INTERFACE I_MotionAxis EXTENDS __SYSTEM.IQueryInterface, 
// 						I_AxisParameters, 
// 						I_AxisStatus, 
// 						I_Home,
// 						I_Halt, 
// 						I_Power, 
// 						I_Reset,
 						I_Output
// 						I_MoveAbsolute,
// 						I_BacklashCompensation

PROPERTY AbortDone : BOOL
GET
END_GET
END_PROPERTY

METHOD AxisEnabled : BOOL
VAR_INPUT
END_VAR
END_METHOD

PROPERTY AxisParamsInit : BOOL
GET
END_GET
END_PROPERTY

PROPERTY AxisState : MC_AxisStates
GET
END_GET
END_PROPERTY

(*
    Handle positive/negative backlash compensation
    User needs to set the direction of backlash from the sign of the compensation value
    Backlash compensation is disabled during referencing (homing).
    When direction is positive/negative, further movement in the negative/positive direction not compensated
    further movement in the negative/positive direction will be compensated
*)
METHOD BacklashCompensation
VAR_INPUT
    Active     : BOOL;
    Compensation	: LREAL;
    RampVelocity	: LREAL;
    DisableMode	: E_DISABLEMODE := E_DISABLEMODE.DisableModeHold;
END_VAR
END_METHOD

(*synced Fbs need just to activate the compensation with a given ramp speed
  other parameters are provided via EPICS (declared in this FB) or via the more extended BackalshCompensation method (simulation) *)
METHOD BacklashCompensationActive
VAR_INPUT
    Active     : BOOL;
    RampVelocity : LREAL;
END_VAR
END_METHOD

{warning 'Add property implementation'}
PROPERTY BacklashCompStatus : BOOL
GET
END_GET
END_PROPERTY

PROPERTY BacklashCompUserEn : BOOL
SET
END_SET
END_PROPERTY

METHOD Halt
VAR_INPUT
	Execute : BOOL;
    Deceleration : LREAL := 0.0;
    Jerk : LREAL := 0.0;
    BufferMode	: MC_BufferMode := MC_BufferMode.MC_Aborting;
END_VAR
END_METHOD

{warning 'Add property implementation'}
PROPERTY HaltActive : BOOL
GET
END_GET
END_PROPERTY

PROPERTY HaltBusy : BOOL
GET
END_GET
END_PROPERTY

PROPERTY HaltDone : BOOL
GET
END_GET
END_PROPERTY

METHOD  Home
VAR_INPUT
	Execute	: BOOL;
	HomeSpeedFast	: LREAL;
	HomeSpeedSlow	: LREAL;
END_VAR
END_METHOD

PROPERTY HomeBusy : BOOL
GET
END_GET
END_PROPERTY

PROPERTY HomeDone : BOOL
GET
END_GET
END_PROPERTY

PROPERTY HomeMode : E_EpicsHomeCmd
GET
END_GET
SET
END_SET
END_PROPERTY

PROPERTY InTargetPosition : BOOL
GET
END_GET
END_PROPERTY

{warning 'Add property implementation'}
PROPERTY MeasureBacklash : LREAL
GET
END_GET
END_PROPERTY

PROPERTY MeasuredAcceleration : LREAL
GET
END_GET
END_PROPERTY

{warning 'Add property implementation'}
PROPERTY MeasuredBacklashComp : LREAL
GET
END_GET
END_PROPERTY

PROPERTY MeasuredPosition : LREAL
GET
END_GET
END_PROPERTY

PROPERTY MeasuredPositionDiff : LREAL
GET
END_GET
END_PROPERTY

PROPERTY MeasuredVelocity : LREAL
GET
END_GET
END_PROPERTY

METHOD MoveAbsolute
VAR_INPUT
    Execute     : BOOL;
    Position	: LREAL;
    Velocity	: LREAL;
    Acceleration	: LREAL := 0.0;
    Deceleration	: LREAL := 0.0;
    Jerk	: LREAL := 0.0;
    BufferMode	: MC_BufferMode := MC_BufferMode.MC_Aborting;
END_VAR
END_METHOD

PROPERTY MoveAbsoluteAborted : BOOL
GET
END_GET
END_PROPERTY

PROPERTY MoveAbsoluteActive : BOOL
GET
END_GET
END_PROPERTY

PROPERTY MoveAbsoluteBusy : BOOL
GET
END_GET
END_PROPERTY

PROPERTY MoveAbsoluteDone : BOOL
GET
END_GET
END_PROPERTY

PROPERTY NegativeMotionIsEnabled : BOOL
GET
END_GET
END_PROPERTY

PROPERTY PositiveMotionIsEnabled : BOOL
GET
END_GET
END_PROPERTY

METHOD Power
VAR_INPUT
    Enable	: BOOL;
    Enable_Positive	: BOOL;
    Enable_Negative	: BOOL;
    Override	: LREAL ;
    BufferMode	: MC_BufferMode;
END_VAR
END_METHOD

PROPERTY PowerActive : BOOL
GET
END_GET
END_PROPERTY

METHOD PowerEnables
VAR_INPUT
    Enable	: BOOL;
    Enable_Positive	: BOOL;
    Enable_Negative	: BOOL;
END_VAR
END_METHOD

PROPERTY PowerIsEnabled : BOOL
GET
END_GET
END_PROPERTY

METHOD Reset
VAR_INPUT
	Execute : BOOL;
END_VAR
END_METHOD

PROPERTY ResetBusy : BOOL
GET
END_GET
END_PROPERTY

PROPERTY ResetDone : BOOL
GET
END_GET
END_PROPERTY

PROPERTY RestoreDone : BOOL
GET
END_GET
END_PROPERTY

PROPERTY SavedPosition : LREAL
GET
END_GET
END_PROPERTY

PROPERTY ScaledEncoderCount : UDINT
GET
END_GET
END_PROPERTY

{warning 'Add property implementation'}
PROPERTY StandStill : BOOL
GET
END_GET
END_PROPERTY

(*
    Check all post condition before updating bCommandedMoveAbsolute
    The implmentatation will depend on the axis type
    DS402 NC/Direct axis : Implementation need to check that the drive is in the correct mode before initaiting the move then set bCommandedMoveAbsolute
    MP NC axis : will immediately write to bCommandedMoveAbsolute
*)
METHOD StartMove : BOOL
VAR_INPUT
    MoveMode	: E_EpicsMotorCmd;
    CmdExecute	: BOOL;
END_VAR
END_METHOD

PROPERTY Stopped : BOOL
GET
END_GET
END_PROPERTY

END_INTERFACE

(* stored: Version 1.1.0.1
   Itf I_MotionAxis: Id {31a902d0-0933-4477-af85-d5a81bbd2467}
   Property AbortDone: Id {5c7662f1-9d2d-42f7-8e24-51d5866c86b3}
   Get Get: Id {93658730-1b85-4a95-9fa2-c21fbe9d7f48}
   Method AxisEnabled: Id {65dbd00d-2aae-4126-bb1b-b72ba759e223}
   Property AxisParamsInit: Id {0ac6452c-b5e1-4e22-865e-3cb2fa5bdfa5}
   Get Get: Id {cf5c8d62-269a-4b22-88e4-cc443108703c}
   Property AxisState: Id {bff14cf8-c54e-4f81-89d2-2b0a7f44eac4}
   Get Get: Id {449be078-56bc-4849-bd3a-e15c9cea95eb}
   Method BacklashCompensation: Id {7436498c-944b-4e18-b9ff-6d68481a3f19}
   Method BacklashCompensationActive: Id {3e7bc661-61f7-4e53-a6c1-341c4d84a32c}
   Property BacklashCompStatus: Id {caf46bd6-b35f-44e4-8914-e70bbd07956d}
   Get Get: Id {f6a45633-a1fa-4659-887f-31976f0aa6aa}
   Property BacklashCompUserEn: Id {94812ccc-d5c4-49f8-aaf1-b91b9d04b484}
   Set Set: Id {84ab6711-b0cf-4074-b1dd-0d70c79947a1}
   Method Halt: Id {c05fa9c9-1bb9-49f8-8b3e-d44f26433d64}
   Property HaltActive: Id {5d6d5bda-e0de-4a28-8aa0-b85c507cdad0}
   Get Get: Id {4f5edcd4-20fe-43f9-8973-d65798036d1c}
   Property HaltBusy: Id {9541a085-e1d1-4a88-8402-724cd91f040a}
   Get Get: Id {8eb7f1c7-9461-46de-8fdb-d396cbb4626b}
   Property HaltDone: Id {a96c6505-72d4-48f7-834a-1162be0cc363}
   Get Get: Id {0d04f02a-d165-4498-8810-653cd0ad98be}
   Method Home: Id {389ec9c0-6958-4b75-bc75-cf73e213180f}
   Property HomeBusy: Id {085e184a-60b7-4e61-b9df-1cb084216a57}
   Get Get: Id {3e4fb446-eba9-4f63-a7ca-7692470d57ec}
   Property HomeDone: Id {180db6b4-ec37-4d47-b243-fc069ef95f8e}
   Get Get: Id {5abbdf75-4945-4b01-8731-586a4b17c65d}
   Property HomeMode: Id {82377409-78bc-42db-8154-8d4d5bb308ee}
   Get Get: Id {1a9eb16b-9f78-44c6-87e2-3304e572b793}
   Set Set: Id {6b7a652e-625f-499d-a110-8ca538ff003d}
   Property InTargetPosition: Id {01bb2d1f-6955-454c-94b8-eb3784e8a966}
   Get Get: Id {616d8ce9-b70c-4636-ad27-5c4193acfb70}
   Property MeasureBacklash: Id {defc67e7-efe7-46f6-b8ce-29d0a4f80c6e}
   Get Get: Id {24364a45-433a-47cd-9268-48134bfc2788}
   Property MeasuredAcceleration: Id {0c6642fb-9a0b-4f3a-b081-4227aa2d097e}
   Get Get: Id {0503172d-53cb-44db-8535-59561f3ebb1d}
   Property MeasuredBacklashComp: Id {5f7b3ef2-d684-40e2-8f28-03dcd8bedbe8}
   Get Get: Id {09fa3778-3e2b-46cd-a257-b54304b0d376}
   Property MeasuredPosition: Id {04c6e978-60d0-4be6-a741-2baf75d815e0}
   Get Get: Id {833856ae-6cd3-4f74-b68e-d04f19c7f43f}
   Property MeasuredPositionDiff: Id {7397084c-0e07-45ab-90f1-aebf1155281f}
   Get Get: Id {1246252f-7184-459d-b216-72ec1b2d0d6b}
   Property MeasuredVelocity: Id {25effada-6d29-4752-b30d-550dfa64e101}
   Get Get: Id {3d2cc533-0f89-444c-abc4-63938ea9897b}
   Method MoveAbsolute: Id {f743ae03-cd9d-4d7e-828a-ea2cf453a8e8}
   Property MoveAbsoluteAborted: Id {85a8c0a8-9a85-40ee-be6b-8e8ac8b6c738}
   Get Get: Id {0385d29c-410c-471c-b9dd-8671da335d2a}
   Property MoveAbsoluteActive: Id {0d4d6e52-7548-45f8-a09c-be5912865edc}
   Get Get: Id {e9c9a3ad-80b4-4ae2-9bf7-80cd6029c39e}
   Property MoveAbsoluteBusy: Id {4df59c3f-7bb2-44c5-bed3-72dbf4fba70e}
   Get Get: Id {9829e242-6925-4891-b633-368ee82fbd1d}
   Property MoveAbsoluteDone: Id {3a920b53-288b-457f-8e2d-a90745ed6e57}
   Get Get: Id {b9e39973-f376-4f69-b7e4-ba733fdf122a}
   Property NegativeMotionIsEnabled: Id {eba716f8-41ff-4e68-81b0-f816ea46fe69}
   Get Get: Id {2a986613-843f-4bcd-b202-f2604e95d197}
   Property PositiveMotionIsEnabled: Id {7341997e-cc82-40d7-a22f-ff83c452b0a2}
   Get Get: Id {6bf8d1d0-42eb-4754-8863-30c805d2aef4}
   Method Power: Id {313af16c-0e71-4ad4-8210-b8ae48a6a0d3}
   Property PowerActive: Id {a296e227-999c-483e-908e-59b8d616bcb1}
   Get Get: Id {96faf1d2-dfba-4184-ba1c-93e82ad5a362}
   Method PowerEnables: Id {b9d13756-5195-47ae-9407-49b1f2466088}
   Property PowerIsEnabled: Id {9699b83a-0072-4b3b-b7ef-6a521cd97971}
   Get Get: Id {57bed3b6-a321-453c-9048-0b175f992ca6}
   Method Reset: Id {45e1cd61-ad60-413b-ade5-3a5bb31fcab7}
   Property ResetBusy: Id {8d74e7a7-96ad-453b-92e4-50c0f920082f}
   Get Get: Id {c1a18b23-e70d-47e7-a3dd-25968fb8461d}
   Property ResetDone: Id {5c15f18a-434c-4360-a939-a0bdc9e0f009}
   Get Get: Id {1b85956f-8d39-43d2-8513-f0014cbfa739}
   Property RestoreDone: Id {4854e4fa-6218-42f7-9a0c-5b2be968b874}
   Get Get: Id {13a18d3e-17f4-4785-85a5-01c8f9059267}
   Property SavedPosition: Id {9d2164dd-1e19-43d4-a6a1-ece31fd9adcb}
   Get Get: Id {a4ad0823-21d1-4852-95b5-b91ce9b1ea7b}
   Property ScaledEncoderCount: Id {ac31d944-ae9d-4416-8ba4-c4a73cec4dfc}
   Get Get: Id {64763161-a809-4119-86c9-c513f284afda}
   Property StandStill: Id {71bf1edc-e05e-4b86-9c40-d2d02284369d}
   Get Get: Id {bf13408a-260d-4106-8122-64c5d13a350e}
   Method StartMove: Id {0cfb7600-869f-45bc-a924-e1dbdd6d1c62}
   Property Stopped: Id {13a1ade1-a2a4-471c-9fd2-4d411b065add}
   Get Get: Id {cb2a6002-931f-4582-ada8-a93edb5b24e4} *)
